// TIA Portal V21 export
TYPE "switchgearHMI"
   STRUCT
      status { S7_SetPoint := 'True'} : Word;
      "step" : USInt;
      stepTime : LTime;
      current : Real;
      alm { S7_SetPoint := 'True'} : Word;
      stopCtx { S7_SetPoint := 'True'} : "stopCtxHMI";
   END_STRUCT;
END_TYPE
